TYPE
    UNI_FanucRobotList :
    UNION
        arFanucRobot : ARRAY[1..2] OF FB_FanucRobot_Basic;
        List         : ST_FanucRobotList;
    END_UNION
END_TYPE

(* stored: Version 1.1.0.1, ProductVersion 3.1.4024.13
   DUT UNI_FanucRobotList: Id {cb52412a-3db2-4978-9a59-b27834506c05} *)
